PROGRAM MoveVirtualAxis
VAR
    currentState : EAxisStates := EAxisStates.Init; // Estado inicial
    nextState : EAxisStates;                        // Próximo estado

    // Variáveis de controle
    axisPosition : LREAL := 0.0;     			// Posição do eixo virtual
    targetPosition : REAL := 1000.0; 			// Posição alvo
    moveSpeed : REAL := 10.0;       			// Velocidade de movimento
    isAxisMoving : BOOL := FALSE;   			// Indicador de movimento
	fb_MoveAbsolutoEixo1: MC_MoveAbsolute;		// Bloco Move Absolute
	fb_MoveAbsolutoEixo2: MC_MoveAbsolute;		// Bloco Move Absolute
	bMoverEixo1Abs: BOOL;						// Aciona o bloco pela primeira vez
	bMoverEixo1Abs2: BOOL;						// Aciona o bloco pela segunda vez
	lrPosicao: LREAL := 1000;
	Timer1: TON;
	Timer2: TON;
	Trigger1: R_TRIG;
	Trigger2: R_TRIG;
	bMoveAbsolutoEixo1Done: BOOL;
	bMoveAbsolutoEixo2Done: BOOL;
END_VAR


CASE currentState OF
    EAxisStates.Init:
        // Inicializa o sistema
        axisPosition := Axes.Axis1.NcToPlc.ActPos;
        isAxisMoving := Axes.Axis1.Status.Moving;
        nextState := EAxisStates.Ready; // Vai para o estado "Ready"
        
    EAxisStates.Ready:
        // Espera o comando para iniciar o movimento
        IF isAxisMoving THEN
            nextState := EAxisStates.Moving; // Se comando recebido, vai para "Moving"
        END_IF

    EAxisStates.Moving:
        // Atualiza a posição do eixo até atingir a posição alvo
        IF axisPosition < targetPosition THEN
            axisPosition := axisPosition + moveSpeed * 0.1; // Atualiza a posição com base na velocidade
        ELSE
            nextState := EAxisStates.Stopped; // Quando atingir o alvo, vai para "Stopped"
        END_IF

    EAxisStates.Stopped:
        // Para o movimento
        isAxisMoving := FALSE;
        nextState := EAxisStates.Ready; // Volta para "Ready" para receber novo comando
END_CASE

// Transição de estados
currentState := nextState;

	//Move Absolute
	fb_MoveAbsolutoEixo1(
		Axis:= Axes.Axis1, 
		Execute:= bMoverEixo1Abs, 
		Position:= lrPosicao, 
		Velocity:= 500.0);
	Trigger1(CLK:= Axes.Axis1.Status.InTargetPosition, Q=> bMoveAbsolutoEixo1Done);
	Timer1(IN:= bMoveAbsolutoEixo1Done, PT:= T#3S, Q=> bMoverEixo1Abs2);
	//Move Absolute
	fb_MoveAbsolutoEixo2(
		Axis:= Axes.Axis1, 
		Execute:= bMoverEixo1Abs2, 
		Position:= 0, 
		Velocity:= 500.0);
	Trigger2(CLK:= fb_MoveAbsolutoEixo2.Busy, Q=> bMoveAbsolutoEixo2Done);
	Timer2(IN:= bMoveAbsolutoEixo2Done, PT:= T#3S, Q=> bMoverEixo1Abs);

END_PROGRAM

(* stored: Version 1.1.0.1, ProductVersion 3.1.4024.13
   POU MoveVirtualAxis: Id {440f1f32-ba99-42b9-b16a-52733d1dfebc}, SpecialFunc None *)
